(*
		2015-06-04	:
			SerialComBuffer
			SerialStringFormat
		2015-06-19	:
			Move SerialStringFormat into the module itself
*)

VAR_GLOBAL
	SerialComBuffer 	: ARRAY [1..MAX_CHANNELS] OF Serial_ComBuffer; 	(*Structure containing the standard buffer variables required for a functioning serial communication. 1 for each channel.*)
END_VAR

(* stored: Version 1.1.0.1, ProductVersion 3.1.0.36
   GVL SerialComm_GVL: Id {f65afae1-2fba-4043-983c-c21e91d2224e} *)
